{attribute 'linkalways'} 
{attribute 'no_explicit_call' := 'This FB is a CLASS and must be accessed using methods or properties'}
{attribute 'enable_dynamic_creation'}
FUNCTION_BLOCK Node_F_VN_MaxElementElementwise_SINT EXTENDS VisionNode
VAR
    ipContainer : _ITcVnContainer;
    nMax : _SINT(0);
    hrPrev : _HRESULT(S_OK);
    hresult : _HRESULT(S_OK);
END_VAR

METHOD PUBLIC  Clone : I_Node
VAR
	pNode : POINTER TO Node_F_VN_MaxElementElementwise_SINT;
END_VAR
pNode := __NEW(Node_F_VN_MaxElementElementwise_SINT);
Clone := pNode^;
END_METHOD

METHOD FB_init : BOOL
VAR_INPUT
	bInitRetains : BOOL; // if TRUE, the retain variables are initialized (warm start / cold start)
	bInCopyCode : BOOL;  // if TRUE, the instance afterwards gets moved into the copy code (online change)
END_VAR
AddInput('ipContainer', ipContainer);
AddInput('hrPrev', hrPrev);
AddOutput('ipContainer', ipContainer);
AddOutput('nMax', nMax);
AddOutput('hresult',hresult);
END_METHOD

METHOD PROTECTED OnExecute
hresult.Value := F_VN_MaxElementElementwise_SINT(
    ipContainer := ipContainer.Value,
    nMax := nMax.Value,
    hrPrev:= hrPrev.Value);
END_METHOD

METHOD PUBLIC PreExecutionCheck
VAR_INPUT
	Check : I_PreExecutionChecks;
END_VAR
Check.IsTrue(ipContainer.IsValid, 'ipContainer must be a valid container');
Check.IsTrue(ipContainer.IsType(TC_GLOBAL_CONST_LIST.ContainerType_Vector_SINT), 'ipContainer contains incorrect type');
END_METHOD

END_FUNCTION_BLOCK

(* stored: Version 1.1.0.1, ProductVersion 3.1.4026.13
   POU Node_F_VN_MaxElementElementwise_SINT: Id {e86e1657-8d4a-4ac6-9791-391da47adb62}, SpecialFunc None
   Folder Constructor: Id {62cc71bf-9331-43a9-8a62-9d745ffb5588}
   Method Clone: Id {20382265-8f10-4470-8a6f-eb0985e2bab6}
   Method FB_init: Id {b919bffe-cb2b-465c-bf77-5f72b9981b3f}
   Method OnExecute: Id {83e302aa-23ed-4cda-98e4-3116ba5d450b}
   Method PreExecutionCheck: Id {71da15b8-0d84-4ff4-89db-54e0c50567cf} *)
